// TIA Portal V17 export
// export: Created 2024-08-07T21:44:12.3547067Z, ExportSetting WithDefaults, DisplayName Totally Integrated Automation Portal, DisplayVersion V17 Update 7, DisplayName TIA Portal Openness, DisplayVersion V17 Update 7, DisplayName TIA Portal Version Control Interface, DisplayVersion V17, DisplayName SINAMICS Startdrive Advanced, DisplayVersion V17 SP2, DisplayName SINAMICS Startdrive G110M, G120, G120C, G120D, G120P, G115D, DisplayVersion V17 SP2, DisplayName SINAMICS Startdrive G130, G150, S120, S150, SINAMICS MV, S210, DisplayVersion V17 SP2, DisplayName STEP 7 Professional, DisplayVersion V17 Update 7, DisplayName STEP 7 Safety, DisplayVersion V17 Update 6, DisplayName WinCC Advanced / Unified PC, DisplayVersion V17 Update 7
VAR_GLOBAL   // PLC tag table "Electronic key system"
   iEksDiagnosticByte AT %IB400 : Byte;   // EKS: Diagnostic byte
   iEksKeyInserted AT %I400.1 : Bool;   // EKS: Key is inserted in reader
   iEksLevel AT %IB401 : Byte;   // EKS: Level
   iEksEmployeeID_1 AT %IB421 : Byte;   // EKS: Employee ID 1
   iEksEmployeeID_2 AT %IB422 : Byte;   // EKS: Employee ID 2
   iEksEmployeeID_3 AT %IB423 : Byte;   // EKS: Employee ID 3
   iEksEmployeeID_4 AT %IB424 : Byte;   // EKS: Employee ID 4
   iEksKeyID_1 AT %IB517 : Byte;   // EKS: Key ID 1
   iEksKeyID_2 AT %IB518 : Byte;   // EKS: Key ID 2
   iEksKeyID_3 AT %IB519 : Byte;   // EKS: Key ID 3
   iEksKeyID_4 AT %IB520 : Byte;   // EKS: Key ID 4
   iEksKeyID_5 AT %IB521 : Byte;   // EKS: Key ID 5
   iEksKeyID_6 AT %IB522 : Byte;   // EKS: Key ID 6
   iEksKeyID_7 AT %IB523 : Byte;   // EKS: Key ID 7
   iEksKeyID_8 AT %IB524 : Byte;   // EKS: Key ID 8
END_VAR
